ADAPTER L3_AAssignMachine
  (* Standard: 61499-1 *)
  (* Version 0.0, 2008-04-22, EQUEROL, UJI *)
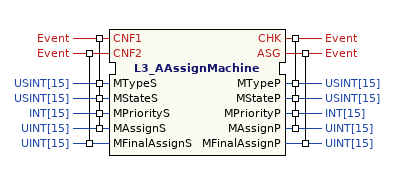
  EVENT_INPUT
    CNF1 WITH MTypeS, MStateS, MPriorityS, MAssignS; (* Confirmation from socket to check request *)
    CNF2 WITH MFinalAssignS; (* Confirmation from socket to assign request *)
  END_EVENT
  EVENT_OUTPUT
    CHK WITH MTypeP, MStateP, MPriorityP, MAssignP; (* Plugin request to check needed machines *)
    ASG WITH MFinalAssignP; (* Plugin request to assign machines to the process plans *)
  END_EVENT
  VAR_INPUT
    MTypeS : ARRAY [0..14] OF USINT; (* Machine Type vector *)
    MStateS : ARRAY [0..14] OF USINT; (* Machine state vector *)
    MPriorityS : ARRAY [0..14] OF INT; (* Machine allocations priority vector *)
    MAssignS : ARRAY [0..14] OF UINT; (* Machine-PP assignation vector *)
    MFinalAssignS : ARRAY [0..14] OF UINT; (* Machine-PP assignation vector *)
  END_VAR
  VAR_OUTPUT
    MTypeP : ARRAY [0..14] OF USINT; (* Machine Type vector *)
    MStateP : ARRAY [0..14] OF USINT; (* Machine State vector *)
    MPriorityP : ARRAY [0..14] OF INT; (* Machine allocations priority vector *)
    MAssignP : ARRAY [0..14] OF UINT; (* Machine-PP assignation vector *)
    MFinalAssignP : ARRAY [0..14] OF UINT; (* Machine-PP Assignation vector *)
  END_VAR
  SERVICE SOCKET/PLUG
    SEQUENCE request_confirm
      SOCKET.REQ(REQD) -> PLUG.REQ(REQD);
      PLUG.CNF(CNFD) -> SOCKET.CNF(CNFD);
    END_SEQUENCE
    SEQUENCE indication_response
      PLUG.IND(INDD) -> SOCKET.IND(INDD);
      SOCKET.RSP(RSPD) -> PLUG.RSP(RSPD);
    END_SEQUENCE
  END_SERVICE
END_ADAPTER
